// TIA Portal project "3M-2n" (V16)

(* hardware
DEVICE "S7-1200 station_1"  S7-1200 Station
   slot 0: "Rack_0"  S7-1200 Rack  Rack  V1.0
   slot 1: "PLC_1"  CPU 1212C AC/DC/Rly  6ES7 212-1BE40-0XB0  V4.0
*)

// ===== PLC "PLC_1"  CPU 1212C AC/DC/Rly =====

VAR_GLOBAL   // PLC tag table "Default tag table"
   "start" AT %I0.0 : Bool;
   "km1" AT %Q0.0 : Bool;
   "km2" AT %Q0.1 : Bool;
   "km3" AT %Q0.2 : Bool;
   "Tag_1" AT %M0.0 : Bool;
   "Tag_2" AT %M0.1 : Bool;
   "Tag_3" AT %M0.2 : Bool;
   "Tag_4" AT %M0.3 : Bool;
   "Tag_5" AT %M0.4 : Bool;
   "Tag_9" AT %M0.6 : Bool;
   "Tag_8" AT %M0.5 : Bool;
   "Tag_6" AT %M0.7 : Bool;
   "Tag_7" AT %M1.0 : Bool;
   "Tag_10" AT %M1.1 : Bool;
   "Tag_11" AT %M1.2 : Bool;
   "Tag_12" AT %M1.3 : Bool;
   "Tag_13" AT %M1.4 : Bool;
   "Tag_14" AT %M1.5 : Bool;
END_VAR

// folder: System blocks/Program resources

DATA_BLOCK "C"   // DB1
{ S7_Optimized_Access := 'TRUE' }
AUTHOR : Simatic
FAMILY : IEC
NAME : CNTR
VERSION : 1.0
// stored: InstanceOfName IEC_COUNTER
"IEC_COUNTER"
BEGIN
END_DATA_BLOCK

DATA_BLOCK "T"   // DB2
{ S7_Optimized_Access := 'TRUE' }
AUTHOR : Simatic
FAMILY : IEC
NAME : IEC_TMR
VERSION : 1.0
// stored: InstanceOfName IEC_TIMER
"IEC_TIMER"
BEGIN
END_DATA_BLOCK

// folder: (top level)

ORGANIZATION_BLOCK "Main"   // OB1, LAD, ProgramCycle
TITLE = "Main Program Sweep (Cycle)"
{ S7_Optimized_Access := 'TRUE' }
VERSION : 0.1
   VAR_INPUT
      Initial_Call : Bool;   // Initial call of this OB
      Remanence : Bool;   // =True, if remanent data are available
   END_VAR
   VAR_TEMP   // added for the SCL form of the ladder/FBD networks
      _w1 : Bool;
      _w2 : Bool;
      _w3 : Bool;
      _w4 : Bool;
      _w5 : Bool;
   END_VAR
BEGIN

REGION Network 1
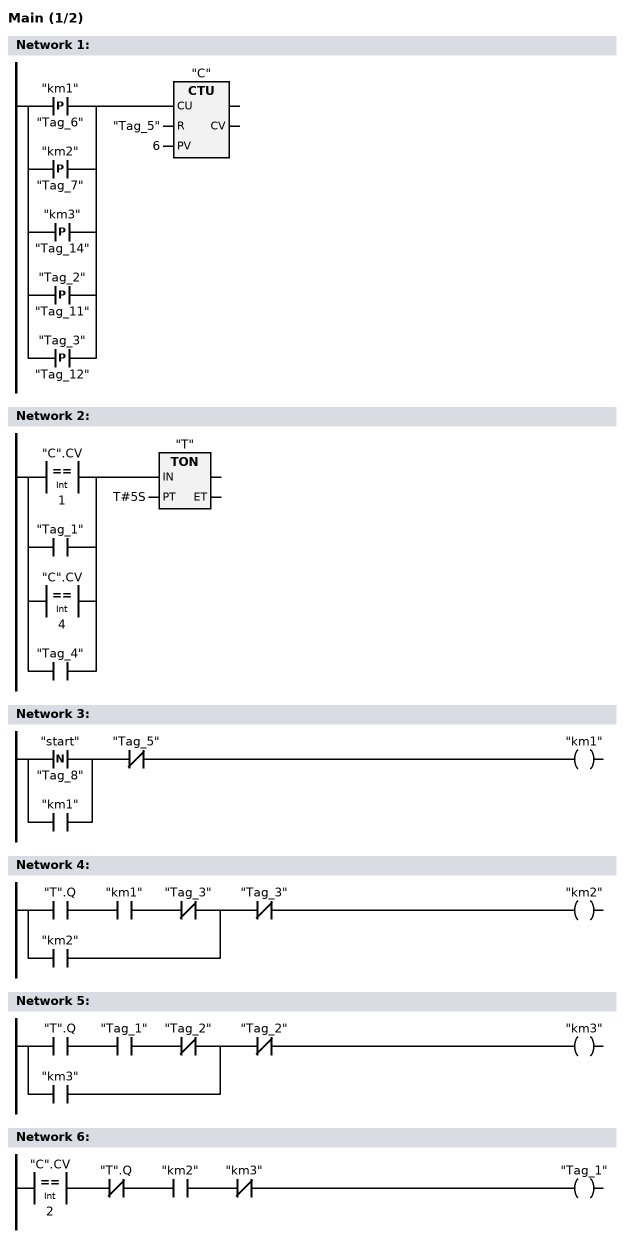
   #_w1 := "km1" AND NOT "Tag_6";   // rising edge of "km1"
   "Tag_6" := "km1";
   #_w2 := "km2" AND NOT "Tag_7";   // rising edge of "km2"
   "Tag_7" := "km2";
   #_w3 := "km3" AND NOT "Tag_14";   // rising edge of "km3"
   "Tag_14" := "km3";
   #_w4 := "Tag_2" AND NOT "Tag_11";   // rising edge of "Tag_2"
   "Tag_11" := "Tag_2";
   #_w5 := "Tag_3" AND NOT "Tag_12";   // rising edge of "Tag_3"
   "Tag_12" := "Tag_3";
   "C".CTU(CU := #_w1 OR #_w2 OR #_w3 OR #_w4 OR #_w5, R := "Tag_5", PV := 6);
END_REGION

REGION Network 2
   "T".TON(IN := ("C".CV = 1) OR "Tag_1" OR ("C".CV = 4) OR "Tag_4", PT := T#5S);
END_REGION

REGION Network 3
   RUNG wire#powerrail
      N_Contact(operand := "start", bit := "Tag_8")
      wire#w1
      I_Contact( "Tag_5" )
      Coil( "km1" )
   END_RUNG
   RUNG wire#powerrail
      Contact( "km1" )
   END_RUNG wire#w1
   // the same network as SCL:
   #_w1 := NOT "start" AND "Tag_8";   // falling edge of "start"
   "Tag_8" := "start";
   "km1" := (#_w1 OR "km1") AND NOT "Tag_5";
END_REGION

REGION Network 4
   RUNG wire#powerrail
      Contact( "T".Q )
      Contact( "km1" )
      I_Contact( "Tag_3" )
      wire#w1
      I_Contact( "Tag_3" )
      Coil( "km2" )
   END_RUNG
   RUNG wire#powerrail
      Contact( "km2" )
   END_RUNG wire#w1
   // the same network as SCL:
   "km2" := (("T".Q AND "km1" AND NOT "Tag_3") OR "km2") AND NOT "Tag_3";
END_REGION

REGION Network 5
   RUNG wire#powerrail
      Contact( "T".Q )
      Contact( "Tag_1" )
      I_Contact( "Tag_2" )
      wire#w1
      I_Contact( "Tag_2" )
      Coil( "km3" )
   END_RUNG
   RUNG wire#powerrail
      Contact( "km3" )
   END_RUNG wire#w1
   // the same network as SCL:
   "km3" := (("T".Q AND "Tag_1" AND NOT "Tag_2") OR "km3") AND NOT "Tag_2";
END_REGION

REGION Network 6
   RUNG wire#powerrail
      { S7_Templates := "SrcType := Int" } EQ_Contact(in1 := "C".CV, in2 := 2)
      I_Contact( "T".Q )
      Contact( "km2" )
      I_Contact( "km3" )
      Coil( "Tag_1" )
   END_RUNG
   // the same network as SCL:
   "Tag_1" := ("C".CV = 2) AND NOT "T".Q AND "km2" AND NOT "km3";
END_REGION

REGION Network 7
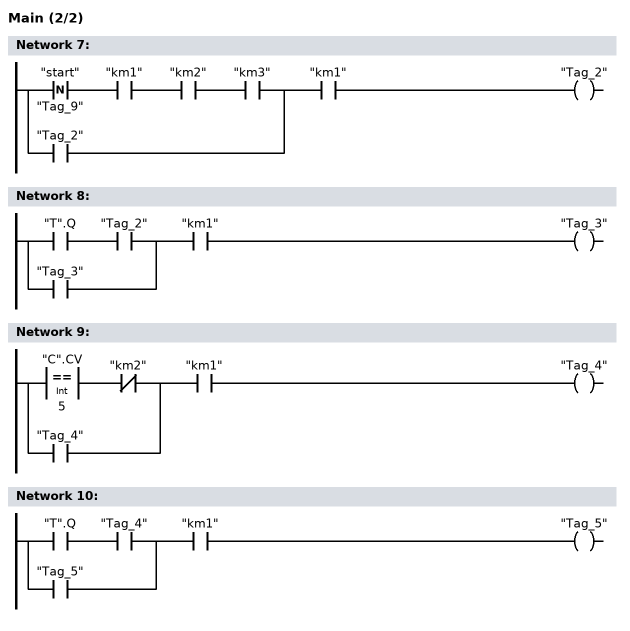
   RUNG wire#powerrail
      N_Contact(operand := "start", bit := "Tag_9")
      Contact( "km1" )
      Contact( "km2" )
      Contact( "km3" )
      wire#w1
      Contact( "km1" )
      Coil( "Tag_2" )
   END_RUNG
   RUNG wire#powerrail
      Contact( "Tag_2" )
   END_RUNG wire#w1
   // the same network as SCL:
   #_w1 := NOT "start" AND "Tag_9";   // falling edge of "start"
   "Tag_9" := "start";
   "Tag_2" := ((#_w1 AND "km1" AND "km2" AND "km3") OR "Tag_2") AND "km1";
END_REGION

REGION Network 8
   RUNG wire#powerrail
      Contact( "T".Q )
      Contact( "Tag_2" )
      wire#w1
      Contact( "km1" )
      Coil( "Tag_3" )
   END_RUNG
   RUNG wire#powerrail
      Contact( "Tag_3" )
   END_RUNG wire#w1
   // the same network as SCL:
   "Tag_3" := (("T".Q AND "Tag_2") OR "Tag_3") AND "km1";
END_REGION

REGION Network 9
   RUNG wire#powerrail
      { S7_Templates := "SrcType := Int" } EQ_Contact(in1 := "C".CV, in2 := 5)
      I_Contact( "km2" )
      wire#w1
      Contact( "km1" )
      Coil( "Tag_4" )
   END_RUNG
   RUNG wire#powerrail
      Contact( "Tag_4" )
   END_RUNG wire#w1
   // the same network as SCL:
   "Tag_4" := ((("C".CV = 5) AND NOT "km2") OR "Tag_4") AND "km1";
END_REGION

REGION Network 10
   RUNG wire#powerrail
      Contact( "T".Q )
      Contact( "Tag_4" )
      wire#w1
      Contact( "km1" )
      Coil( "Tag_5" )
   END_RUNG
   RUNG wire#powerrail
      Contact( "Tag_5" )
   END_RUNG wire#w1
   // the same network as SCL:
   "Tag_5" := (("T".Q AND "Tag_4") OR "Tag_5") AND "km1";
END_REGION
END_ORGANIZATION_BLOCK